// TIA Portal V17 export
// export: Created 2025-03-10T13:13:16.7402002Z, ExportSetting WithDefaults, DisplayName Totally Integrated Automation Portal, DisplayVersion V17 Update 8, DisplayName TIA Portal Openness, DisplayVersion V17 Update 8, DisplayName TIA Portal Version Control Interface, DisplayVersion V17, DisplayName SINAMICS Startdrive Advanced, DisplayVersion V17 SP2, DisplayName SINAMICS Startdrive G110M, G120, G120C, G120D, G120P, G115D, DisplayVersion V17 SP2, DisplayName SINAMICS Startdrive G130, G150, S120, S150, SINAMICS MV, S210, DisplayVersion V17 SP2, DisplayName STEP 7 Professional, DisplayVersion V17 Update 8, DisplayName SINUMERIK ONE STEP 7 Toolbox, DisplayVersion V17 Update 12, DisplayName SINUMERIK 840D sl STEP 7 Toolbox, DisplayVersion V17 Update 12, DisplayName STEP 7 Safety, DisplayVersion V17 Update 6, DisplayName WinCC Advanced, DisplayVersion V17 Update 8
DATA_BLOCK "DB2200_NETWORKS_STATE"   // DB2200
{ S7_Optimized_Access := 'FALSE'; DB_Accessible_From_OPC_UA := 'FALSE' }
AUTHOR : ETXETAR
VERSION : 1.0
// stored: AutoNumber false, DBAccessibleFromOPCUA false, DBAccessibleFromWebserver true, IsOnlyStoredInLoadMemory false, IsWriteProtectedInAS false
   VAR RETAIN
      myMode : UInt := 2;
      ReturnValue : Word;
      SUPPRESS_PROFIBUS_SLAVE : Array[1..1023] of Bool;   // SUPPRESS PROFIBUS SLAVE
      FAULT_IN_PROFIBUS_SLAVE : Array[0..1023] of Bool;   // FAULT IN PROFIBUS SLAVE
      SUPPRESS_PROFINET_SLAVE : Array[1..1023] of Bool;   // SUPPRESS PROFINET SLAVE
      FAULT_IN_PROFINET_SLAVE : Array[0..1023] of Bool;   // FAULT IN PROFINET SLAVE
      PROFIBUS_IS_ALARMS : Bool;   // IMMEDIATE STOP ALARM FOR PROFIBUS NETWORK / PROFIBUS IMMEDIATE STOP ALARMS
      PROFIBUS_SEOC_ALARMS : Bool;   // STOP END OF CYCLE ALARM FOR PROFIBUS NETWORK / PROFIBUS STOP END OF CYCLE ALARMS
      PROFIBUS_RHP_SEOC_ALARMS : Bool;   // RETURN HOME POSITION & STOP END OF CYCLE ALARM FOR PROFIBUS NETWORK / PROFIBUS RETURN HOME POSITION AND STOP END OF CYCLE ALARMS
      PROFINET_IS_ALARMS : Bool;   // IMMEDIATE STOP ALARM FOR PROFINET NETWORK / PROFINET IMMEDIATE STOP ALARMS
      PROFINET_SEOC_ALARMS : Bool;   // STOP END OF CYCLE ALARM FOR PROFINET NETWORK / PROFINET STOP END OF CYCLE ALARMS
      PROFINET_RHP_SEOC_ALARMS : Bool;   // RETURN HOME POSITION & STOP END OF CYCLE ALARM FOR PROFINET NETWORK / PROFINET RETURN HOME POSITION AND STOP END OF CYCLE ALARMS
      TIMER_SUPPRESS_PROFIBUS_SLAVES { S7_SetPoint := 'True'} : TOF_TIME;   // SUPPRESS PROFIBUS SLAVE TIMER
      TIMER_SUPPRESS_PROFINET_SLAVES { S7_SetPoint := 'True'} : TOF_TIME;   // SUPPRESS PROFINET SLAVE TIMER
   END_VAR
BEGIN
   TIMER_SUPPRESS_PROFIBUS_SLAVES.PT := T#10s;
   TIMER_SUPPRESS_PROFINET_SLAVES.PT := T#10s;
END_DATA_BLOCK
